{attribute 'qualified_only'}
VAR_GLOBAL
  Com : ZCom;
END_VAR
VAR_GLOBAL PERSISTENT
  Data : ZData;
END_VAR

(* stored: Version 1.1.0.1
   GVL ZGlobal: Id {eb156a20-0182-495f-b441-a766648df103} *)
